FUNCTION_BLOCK FB_DRIVE_TEST EXTENDS TcUnit.FB_TestSuite
VAR_INPUT
END_VAR
VAR_OUTPUT
END_VAR
VAR
END_VAR

SteerAngleTest();
DiffDriveTest();

METHOD DiffDriveTest : REFERENCE TO FB_Test
VAR
	
END_VAR
TEST('DifferentialDriveTest');



TEST_FINISHED();
END_METHOD

METHOD SteerAngleTest : REFERENCE TO FB_Test
VAR
	Drive	: FB_DRIVE;
	AngleInput			: LREAL := 45;
	LeftAngleCalc		: LREAL;
	RightAngleCalc		: LREAL;	
	LeftAngleExpected	: LREAL := 38.89;
	RightAngleExpected	: LREAL := 51.03;
END_VAR
TEST('SteerAngleTest');

(*Zero Steering Angle*)
Drive.CalcWheelAngle(0);
LeftAngleCalc := Drive.SteerLeftAngleTest;
RightAngleCalc := Drive.SteerRightAngleTest;
			
AssertEquals_LREAL(Expected := 0,
				Actual := LeftAngleCalc,
				Delta := 0.1,
				Message := 'Left Angle 0 Calculation Incorrect');
				
AssertEquals_LREAL(Expected := 0,
				Actual := RightAngleCalc,
				Delta := 0.1,
				Message := 'Right Angle 0 Calculation Incorrect');

(*45 Degree Steering Angle*)				
Drive.CalcWheelAngle(AngleInput);
LeftAngleCalc := Drive.SteerLeftAngleTest;
RightAngleCalc := Drive.SteerRightAngleTest;

AssertEquals_LREAL(Expected := LeftAngleExpected,
				Actual := LeftAngleCalc,
				Delta := 0.1,
				Message := 'Left Angle 45 Calculation Incorrect');
				
AssertEquals_LREAL(Expected := RightAngleExpected,
				Actual := RightAngleCalc,
				Delta := 0.1,
				Message := 'Right Angle 45 Calculation Incorrect');

(*-45 Degree Steering Angle*)			
Drive.CalcWheelAngle(-AngleInput);
LeftAngleCalc := Drive.SteerLeftAngleTest;
RightAngleCalc := Drive.SteerRightAngleTest;

AssertEquals_LREAL(Expected := -RightAngleExpected,
				Actual := LeftAngleCalc,
				Delta := 0.1,
				Message := 'Left Angle -45 Calculation Incorrect');
				
AssertEquals_LREAL(Expected := -LeftAngleExpected,
				Actual := RightAngleCalc,
				Delta := 0.1,
				Message := 'Right Angle -45 Calculation Incorrect');
				
(*Positive Max Steering Angle*)

(*Negative Max Steering Angle*)

(*Positive Out of Range Steering Angle*)

(*Negative Out of Range Steering Angle*)
			
TEST_FINISHED();
END_METHOD

END_FUNCTION_BLOCK

(* stored: Version 1.1.0.1, ProductVersion 3.1.4024.12
   POU FB_DRIVE_TEST: Id {5ef7f248-2813-4803-9c60-282f0431de80}, SpecialFunc None
   Method DiffDriveTest: Id {2ddda7bd-148f-4d06-9902-cc6fa47938b4}
   Method SteerAngleTest: Id {c51523c3-14fd-4809-a98e-7fb50e3f3285} *)
